PROGRAM PRG_HOMMING
VAR
END_VAR

END_PROGRAM

(* stored: Version 1.1.0.1, ProductVersion 3.1.4024.12
   POU PRG_HOMMING: Id {e2c004dd-dc4e-4568-9713-155f8b0cd73c}, SpecialFunc None *)
